// TIA Portal V18 export
FUNCTION_BLOCK "DataLogging"   // FB4, LAD
{ S7_Optimized_Access := 'TRUE' }
VERSION : 0.1
// stored: AutoNumber true, IsIECCheckEnabled false, IsRetainMemResEnabled false, MemoryReserve 100, SetENOAutomatically false, UDAEnableTagReadback false
   VAR_INPUT
      CreateFile : Bool;
      StartLogging : Bool;
      Variable01in_Bool : Bool;
      Name_01 : String;
      Variable02in_Bool : Bool;
      Name_02 : String;
      Variable03in_Dint : DInt;
      Name_03 : String;
      Variable04in_Dint : DInt;
      Name_04 : String;
      Variable05in_Dint : DInt;
      Name_05 : String;
      Variable06in_Dint : DInt;
      Name_06 : String;
   END_VAR
   VAR_OUTPUT
      Variable01out_Bool : Bool;
      Variable02out_Bool : Bool;
      Variable03out_Dint : DInt;
      Variable04out_Dint : DInt;
      Variable05out_Dint : DInt;
      Variable06out_Dint : DInt;
      LogColumns : String;
   END_VAR
   VAR
      FileName : String := 'Logging_Test_01';
      REQ : Bool;
      ID : DWord;
      StartingTime : DTL;
      ReturnValue : Int;
      AmountOfRecords : UDInt := 10000;   // For 864000 and 10 records per sec = 24h
      StartLoggingM : Bool;
      WriteColumn : Int;
      Column01Internal { ExternalAccessible := 'False'; ExternalVisible := 'False'; ExternalWritable := 'False'} : String;
      Column02Internal { ExternalAccessible := 'False'; ExternalVisible := 'False'; ExternalWritable := 'False'} : String;
      Column03Internal { ExternalAccessible := 'False'; ExternalVisible := 'False'; ExternalWritable := 'False'} : String;
      Column04Internal { ExternalAccessible := 'False'; ExternalVisible := 'False'; ExternalWritable := 'False'} : String;
      Column05Internal : String;
      Column06Internal : String;
      WriteColumnReady : Bool;
      RecordCount : DInt;
   END_VAR
   VAR CONSTANT
      NameOfColumn01 : String := 'TestColumn_01';
      NameOfColumn02 : String := 'TestColumn_02';
   END_VAR
   VAR_TEMP   // added for the SCL form of the ladder/FBD networks
      _w1 : Bool;
      _w2 : Bool;
      _w3 : Bool;
      _w4 : Bool;
      _w5 : Bool;
   END_VAR
BEGIN

REGION Network 1: Start logging
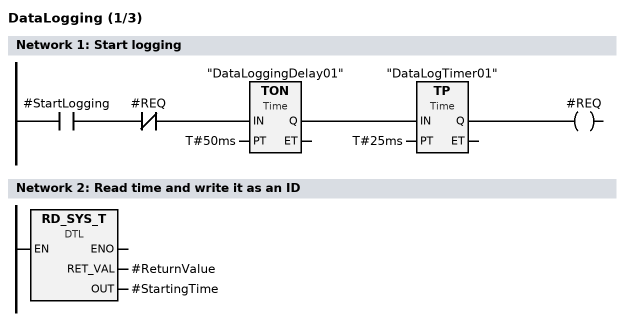
   RUNG wire#powerrail
      Contact( #StartLogging )
      I_Contact( #REQ )
      { S7_Templates := "time_type := Time" } "DataLoggingDelay01".TON(pt := T#50ms, et =>)
      { S7_Templates := "time_type := Time" } "DataLogTimer01".TP(pt := T#25ms, et =>)
      Coil( #REQ )
   END_RUNG
   // the same network as SCL:
   "DataLoggingDelay01".TON(IN := #StartLogging AND NOT #REQ, PT := T#50ms);
   "DataLogTimer01".TP(IN := "DataLoggingDelay01".Q, PT := T#25ms);
   #REQ := "DataLogTimer01".Q;
END_REGION

REGION Network 2: Read time and write it as an ID
   RUNG wire#powerrail
      { S7_Templates := "date_type := DTL" } RD_SYS_T(RET_VAL => #ReturnValue, OUT => #StartingTime)
   END_RUNG
   // the same network as SCL:
   #ReturnValue := RD_SYS_T(OUT => #StartingTime);
END_REGION

REGION Network 3: Write Column Names
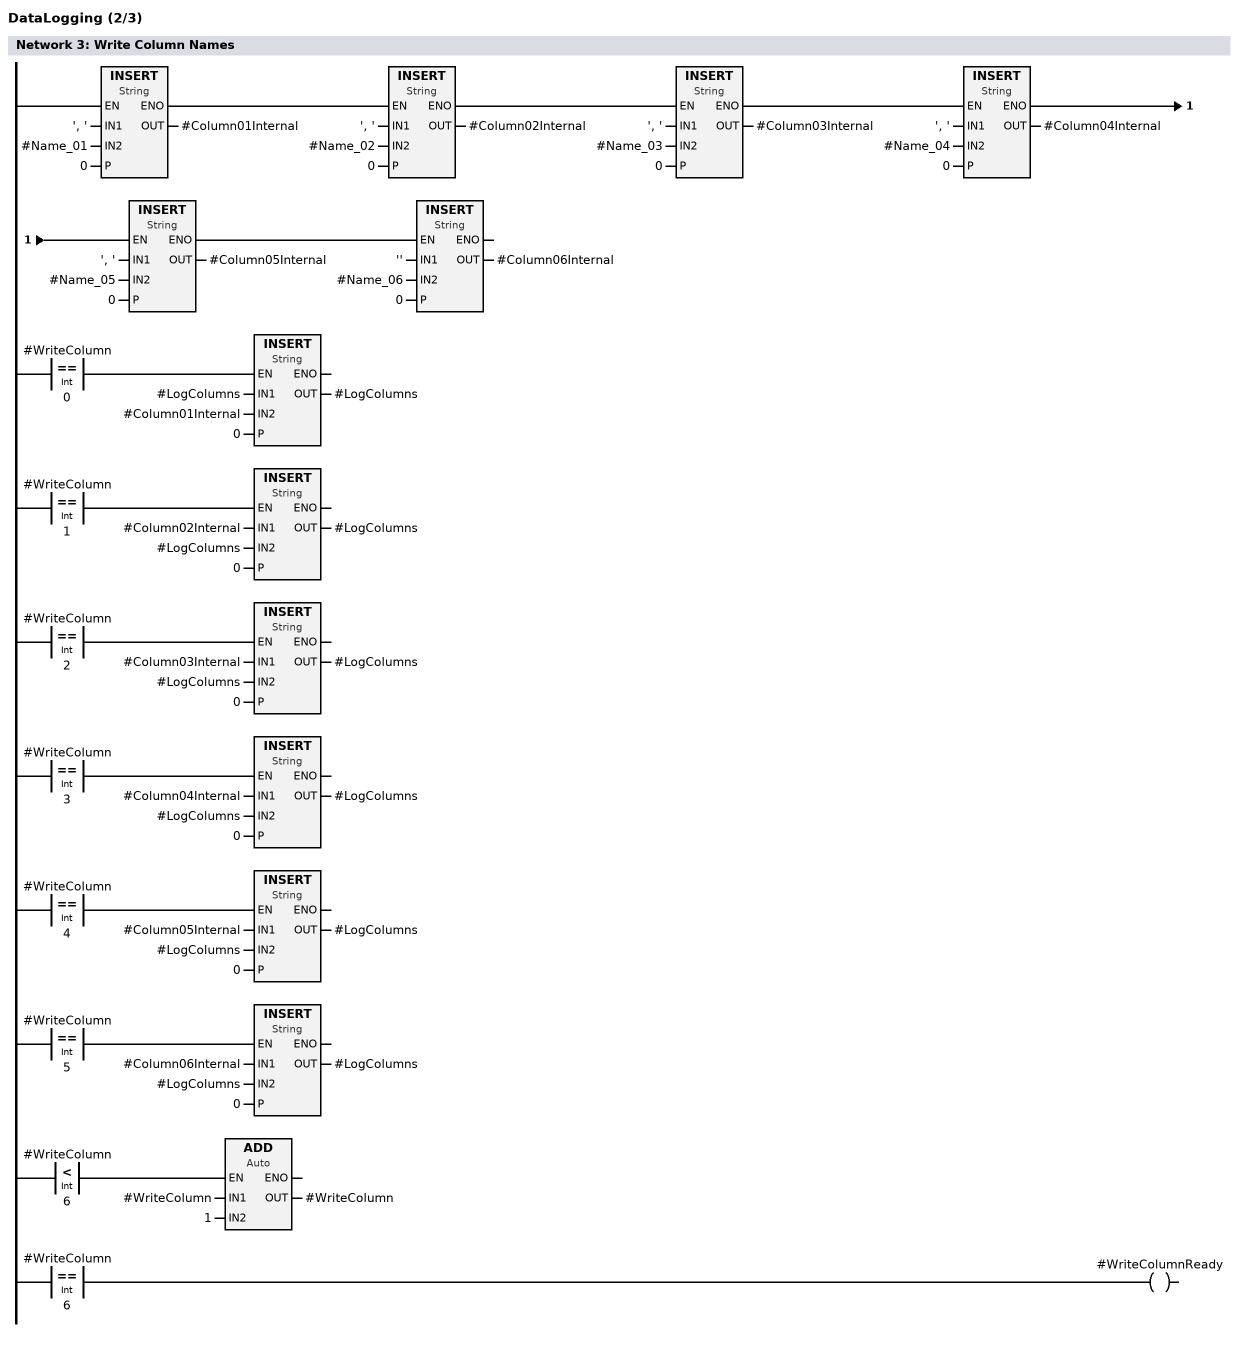
   RUNG wire#powerrail
      { S7_Templates := "str_type := String" } INSERT(IN1 := ', ', IN2 := #Name_01, P := 0, OUT => #Column01Internal)
      { S7_Templates := "str_type := String" } INSERT(IN1 := ', ', IN2 := #Name_02, P := 0, OUT => #Column02Internal)
      { S7_Templates := "str_type := String" } INSERT(IN1 := ', ', IN2 := #Name_03, P := 0, OUT => #Column03Internal)
      { S7_Templates := "str_type := String" } INSERT(IN1 := ', ', IN2 := #Name_04, P := 0, OUT => #Column04Internal)
      { S7_Templates := "str_type := String" } INSERT(IN1 := ', ', IN2 := #Name_05, P := 0, OUT => #Column05Internal)
      { S7_Templates := "str_type := String" } INSERT(IN1 := '', IN2 := #Name_06, P := 0, OUT => #Column06Internal)
   END_RUNG
   RUNG wire#powerrail
      { S7_Templates := "SrcType := Int" } EQ_Contact(in1 := #WriteColumn, in2 := 0)
      { S7_Templates := "str_type := String" } INSERT(IN1 := #LogColumns, IN2 := #Column01Internal, P := 0, OUT => #LogColumns)
   END_RUNG
   RUNG wire#powerrail
      { S7_Templates := "SrcType := Int" } EQ_Contact(in1 := #WriteColumn, in2 := 1)
      { S7_Templates := "str_type := String" } INSERT(IN1 := #Column02Internal, IN2 := #LogColumns, P := 0, OUT => #LogColumns)
   END_RUNG
   RUNG wire#powerrail
      { S7_Templates := "SrcType := Int" } EQ_Contact(in1 := #WriteColumn, in2 := 2)
      { S7_Templates := "str_type := String" } INSERT(IN1 := #Column03Internal, IN2 := #LogColumns, P := 0, OUT => #LogColumns)
   END_RUNG
   RUNG wire#powerrail
      { S7_Templates := "SrcType := Int" } EQ_Contact(in1 := #WriteColumn, in2 := 3)
      { S7_Templates := "str_type := String" } INSERT(IN1 := #Column04Internal, IN2 := #LogColumns, P := 0, OUT => #LogColumns)
   END_RUNG
   RUNG wire#powerrail
      { S7_Templates := "SrcType := Int" } EQ_Contact(in1 := #WriteColumn, in2 := 4)
      { S7_Templates := "str_type := String" } INSERT(IN1 := #Column05Internal, IN2 := #LogColumns, P := 0, OUT => #LogColumns)
   END_RUNG
   RUNG wire#powerrail
      { S7_Templates := "SrcType := Int" } EQ_Contact(in1 := #WriteColumn, in2 := 5)
      { S7_Templates := "str_type := String" } INSERT(IN1 := #Column06Internal, IN2 := #LogColumns, P := 0, OUT => #LogColumns)
   END_RUNG
   RUNG wire#powerrail
      { S7_Templates := "SrcType := Int" } LT_Contact(in1 := #WriteColumn, in2 := 6)
      Add(in1 := #WriteColumn, in2 := 1, out => #WriteColumn)
   END_RUNG
   RUNG wire#powerrail
      { S7_Templates := "SrcType := Int" } EQ_Contact(in1 := #WriteColumn, in2 := 6)
      Coil( #WriteColumnReady )
   END_RUNG
   // the same network as SCL:
   INSERT(IN1 := ', ', IN2 := #Name_01, P := 0, OUT => #Column01Internal, ENO => #_w1);
   INSERT(EN := #_w1, IN1 := ', ', IN2 := #Name_02, P := 0, OUT => #Column02Internal, ENO => #_w2);
   INSERT(EN := #_w2, IN1 := ', ', IN2 := #Name_03, P := 0, OUT => #Column03Internal, ENO => #_w3);
   INSERT(EN := #_w3, IN1 := ', ', IN2 := #Name_04, P := 0, OUT => #Column04Internal, ENO => #_w4);
   INSERT(EN := #_w4, IN1 := ', ', IN2 := #Name_05, P := 0, OUT => #Column05Internal, ENO => #_w5);
   IF #_w5 THEN INSERT(IN1 := '', IN2 := #Name_06, P := 0, OUT => #Column06Internal); END_IF;
   IF #WriteColumn = 0 THEN
       INSERT(IN1 := #LogColumns, IN2 := #Column01Internal, P := 0, OUT => #LogColumns);
   END_IF;
   IF #WriteColumn = 1 THEN
       INSERT(IN1 := #Column02Internal, IN2 := #LogColumns, P := 0, OUT => #LogColumns);
   END_IF;
   IF #WriteColumn = 2 THEN
       INSERT(IN1 := #Column03Internal, IN2 := #LogColumns, P := 0, OUT => #LogColumns);
   END_IF;
   IF #WriteColumn = 3 THEN
       INSERT(IN1 := #Column04Internal, IN2 := #LogColumns, P := 0, OUT => #LogColumns);
   END_IF;
   IF #WriteColumn = 4 THEN
       INSERT(IN1 := #Column05Internal, IN2 := #LogColumns, P := 0, OUT => #LogColumns);
   END_IF;
   IF #WriteColumn = 5 THEN
       INSERT(IN1 := #Column06Internal, IN2 := #LogColumns, P := 0, OUT => #LogColumns);
   END_IF;
   IF #WriteColumn < 6 THEN #WriteColumn := #WriteColumn + 1; END_IF;
   #WriteColumnReady := #WriteColumn = 6;
END_REGION

REGION Network 4: Data Logging Transfer
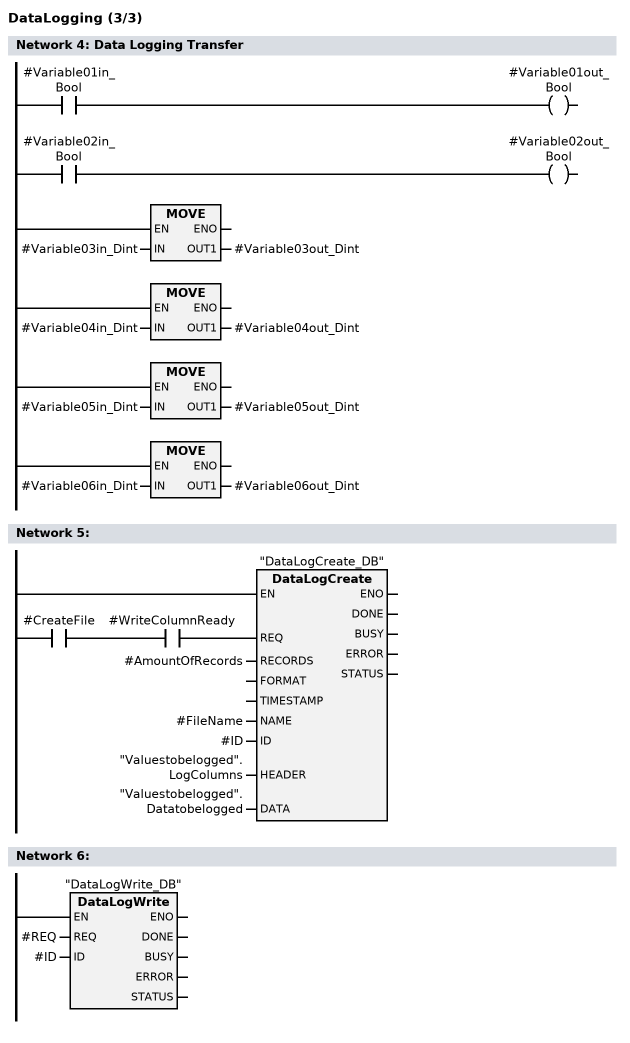
   RUNG wire#powerrail
      Contact( #Variable01in_Bool )
      Coil( #Variable01out_Bool )
   END_RUNG
   RUNG wire#powerrail
      Contact( #Variable02in_Bool )
      Coil( #Variable02out_Bool )
   END_RUNG
   RUNG wire#powerrail
      Move(in := #Variable03in_Dint, out1 => #Variable03out_Dint)
   END_RUNG
   RUNG wire#powerrail
      Move(in := #Variable04in_Dint, out1 => #Variable04out_Dint)
   END_RUNG
   RUNG wire#powerrail
      Move(in := #Variable05in_Dint, out1 => #Variable05out_Dint)
   END_RUNG
   RUNG wire#powerrail
      Move(in := #Variable06in_Dint, out1 => #Variable06out_Dint)
   END_RUNG
   // the same network as SCL:
   #Variable01out_Bool := #Variable01in_Bool;
   #Variable02out_Bool := #Variable02in_Bool;
   #Variable03out_Dint := #Variable03in_Dint;
   #Variable04out_Dint := #Variable04in_Dint;
   #Variable05out_Dint := #Variable05in_Dint;
   #Variable06out_Dint := #Variable06in_Dint;
END_REGION

REGION Network 5
   RUNG wire#powerrail
      "DataLogCreate_DB".DataLogCreate(REQ := wire#w1, RECORDS := #AmountOfRecords, FORMAT :=, TIMESTAMP :=, "NAME" := #FileName, ID := #ID, HEADER := "Valuestobelogged".LogColumns, DATA := "Valuestobelogged".Datatobelogged, DONE =>, BUSY =>, ERROR =>, STATUS =>)
   END_RUNG
   RUNG wire#powerrail
      Contact( #CreateFile )
      Contact( #WriteColumnReady )
   END_RUNG wire#w1
   // the same network as SCL:
   "DataLogCreate_DB"(REQ := #CreateFile AND #WriteColumnReady,   // DataLogCreate
                      RECORDS := #AmountOfRecords,
                      "NAME" := #FileName,
                      ID := #ID,
                      HEADER := "Valuestobelogged".LogColumns,
                      DATA := "Valuestobelogged".Datatobelogged);
END_REGION

REGION Network 6
   RUNG wire#powerrail
      "DataLogWrite_DB".DataLogWrite(REQ := #REQ, ID := #ID, DONE =>, BUSY =>, ERROR =>, STATUS =>)
   END_RUNG
   // the same network as SCL:
   "DataLogWrite_DB"(REQ := #REQ, ID := #ID);   // DataLogWrite
END_REGION
END_FUNCTION_BLOCK
